//{{V2}}
DATA_BLOCK DB10

AUTHOR:mh
FAMILY:nb
NAME:nb
VERSION:1.0


       STRUCT
         b0:REAL
         b1:REAL
         b2:REAL
         b3:REAL
         b4:REAL
         b5:REAL
       END_STRUCT
BEGIN

       b0:=0.000000e+00
       b1:=0.000000e+00
       b2:=0.000000e+00
       b3:=0.000000e+00
       b4:=0.000000e+00
       b5:=0.000000e+00
END_DATA_BLOCK
